FUNCTION_BLOCK FB_Map_QV
VAR_INPUT
END_VAR
VAR_OUTPUT
END_VAR
VAR
	A: stQV_POINT;
	B: stQV_POINT;
	C: stQV_POINT;
	D: stQV_POINT;
	E: stQV_POINT;
	F: stQV_POINT;
	G: stQV_POINT;
	
	max_qv_correction: REAL;
	min_qv_correction: REAL;
	v_ratio: REAL;
	t: REAL;
	i: UINT;
	x: REAL;
	y: REAL;
END_VAR

v_ratio := GVL.VIRTUAL_METER.measured_voltage / GVL_Voltage.reference_value;

/// definizione delle coordiante dei punti della mappa Q/V///
A.q_pnd_ratio := 0;
A.voltage_ratio := 1.1;

B.q_pnd_ratio := 0.30;
B.voltage_ratio := 1.05;

C.q_pnd_ratio := 0.30;
C.voltage_ratio := 0.95;

D.q_pnd_ratio := 0;
D.voltage_ratio := 0.9;

E.q_pnd_ratio := -0.35;
E.voltage_ratio := 0;
/////////////////////////////////////////////////////////////

IF v_ratio > B.voltage_ratio AND v_ratio <= A.voltage_ratio THEN
	min_qv_correction := -0.35;
	t := (v_ratio - A.voltage_ratio) / (A.voltage_ratio - B.voltage_ratio);
	max_qv_correction := t*B.q_pnd_ratio + (1 - t)*A.q_pnd_ratio;
 


ELSIF v_ratio <= B.voltage_ratio AND v_ratio >= C.voltage_ratio THEN
	max_qv_correction := 0.30;
	min_qv_correction := -0.35;



ELSIF v_ratio < C.voltage_ratio AND v_ratio >= D.voltage_ratio THEN
	max_qv_correction := 0.30;
	t := (v_ratio - D.voltage_ratio) / (C.voltage_ratio - D.voltage_ratio);
	min_qv_correction := t*C.q_pnd_ratio + (1 - t)*D.q_pnd_ratio; 
END_IF 


// TO DO: per implementazioni future di una regolazione mediante mappa 
//FOR i := 1 TO GVL_React_Pwr.n_points DO
//	IF v_ratio >= GVL_React_Pwr.enhanced_points[i][1] THEN 
//		x := GVL_React_Pwr.enhanced_points[i][1];
//		y := GVL_React_Pwr.enhanced_points[i][2];
//		g := GVL_React_Pwr.enhanced_points[i][3];
		
//		GVL_Voltage.output_qv_regulation := y + g*(v_ratio - x);
//		EXIT
//	END_IF
//END_FOR


IF GVL_Voltage.output_qv_regulation < min_qv_correction THEN
	GVL_Voltage.output_qv_regulation := min_qv_correction;
END_IF
	
IF GVL_Voltage.output_qv_regulation > max_qv_correction THEN
	GVL_Voltage.output_qv_regulation := max_qv_correction;
END_IF

END_FUNCTION_BLOCK

(* stored: Version 1.1.0.1, ProductVersion 3.1.4026.11
   POU FB_Map_QV: Id {37be17ce-be6c-451d-b406-f197c7e7f39c}, SpecialFunc None *)
